Universal Robots PolyScope program: Bridge_triangle_roof.urp

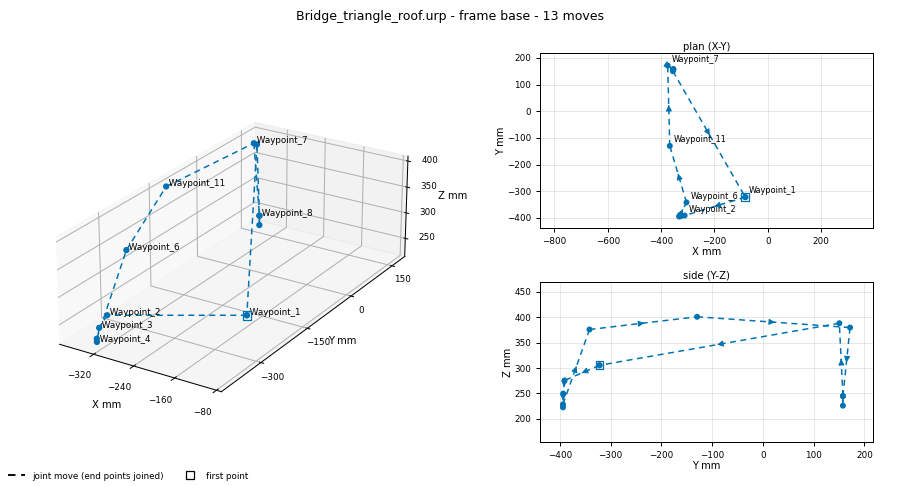
[picture p0: tool path of Bridge_triangle_roof.urp in frame base, 13 of 13 moves have a stored position in this frame; points joined in program order, loops and branches not executed]
Program Bridge_triangle_roof (installation=default directory=/programs/usbdisk/Zahra createdIn=5.11.11.1010533 lastSavedIn=5.11.11.1010533 robotSerialNumber=20205300864)
Calibrated DH parameters: a=[-0.000166, -0.243494, -0.153108, 0.000057, -0.000123, 0]; d=[0.151897, -1.34267, 53.988124, -52.514559, 0.085283, 0.092193]; alpha=[1.572472, -0.003756, 0.002824, 1.570807, -1.572621, 0]; deltaTheta=[0, 0.020704, 7.033215, -0.770746, 0.000004, 0]
Robot Program (runOnlyOnce=true)
  MoveJ speed 60 deg/s, acceleration 80 deg/s^2 (useActiveTCP=true) feature=Base
    Waypoint Waypoint_1: TCP in base x=-84.299 y=-321.875 z=305.481 mm, rx=-2.0809 ry=-2.2572 rz=0.0984 rad; joints [-79.978, -91.201, -87.971, -91.7, 84.671, 815.506] deg
    Waypoint Waypoint_2: TCP in base x=-311.801 y=-390.806 z=275.565 mm, rx=-2.2649 ry=-2.1055 rz=0.1333 rad; joints [-112.548, -138.493, -28.193, -99.813, 85.37, 791.491] deg
    Waypoint Waypoint_3: TCP in base x=-326.771 y=-393.435 z=249.787 mm, rx=2.215 ry=2.2214 rz=-0.0644 rad; joints [-114.765, -143.708, -24.768, -99.132, 89.224, 785.045] deg
    Waypoint Waypoint_4: TCP in base x=-331.937 y=-393.874 z=222.59 mm, rx=2.1803 ry=2.2287 rz=-0.0042 rad; joints [-115.635, -145.452, -28.079, -95.78, 91.072, 783.114] deg
    URCap Gripper (Robotiq_Grippers, Robotiq Inc.) dataModel(position=59.2156862745098, force=94.0, speed=40.0, positionInDouble=59.2156862745098, forceInDouble=94.0, speedInDouble=40.0, slaveIds=[9], blocking=true, robotCompliant=false)
    Waypoint Waypoint_5: TCP in base x=-331.939 y=-393.873 z=228.535 mm, rx=2.1803 ry=2.2287 rz=-0.0043 rad; joints [-115.63, -145.851, -25.689, -97.768, 91.067, 783.115] deg
    Waypoint Waypoint_6: TCP in base x=-304.837 y=-341.621 z=375.948 mm, rx=2.1229 ry=2.1896 rz=-0.3358 rad; joints [-115.077, -126.752, -25.522, -104.372, 89.719, 783.12] deg
    Waypoint Waypoint_11: TCP in base x=-367.481 y=-129.683 z=400.982 mm, rx=-2.0842 ry=-2.3405 rz=-0.0182 rad; joints [-140.769, -116.62, -27.668, -126.196, 89.307, 752.639] deg
    Waypoint Waypoint_7: TCP in base x=-375.414 y=171.565 z=379.774 mm, rx=-2.1093 ry=-2.3182 rz=0.0687 rad; joints [-186.479, -119.065, -31.593, -117.454, 91.662, 708.179] deg
    Waypoint Waypoint_8: TCP in base x=-354.29 y=157.579 z=244.826 mm, rx=-2.2211 ry=-2.2068 rz=0.0358 rad; joints [-184.497, -106.857, -86.723, -75.009, 90.588, 716.008] deg
    Waypoint Waypoint_9: TCP in base x=-354.309 y=157.557 z=225.911 mm, rx=-2.2211 ry=-2.2068 rz=0.0359 rad; joints [-184.501, -108.084, -90.347, -70.153, 90.592, 716.013] deg
    URCap Gripper (Robotiq_Grippers, Robotiq Inc.) dataModel(position=33.72549019607843, force=94.0, speed=40.0, positionInDouble=33.72549019607843, forceInDouble=94.0, speedInDouble=40.0, slaveIds=[9], blocking=true, robotCompliant=false)
    Waypoint Waypoint_8: TCP in base x=-354.29 y=157.579 z=244.826 mm, rx=-2.2211 ry=-2.2068 rz=0.0358 rad; joints [-184.497, -106.857, -86.723, -75.009, 90.588, 716.008] deg
    Waypoint Waypoint_10: TCP in base x=-355.906 y=150.496 z=388.296 mm, rx=-2.1322 ry=-2.1758 rz=0.1564 rad; joints [-183.387, -106.861, -50.233, -105.001, 90.897, 715.571] deg
    Waypoint Waypoint_1: TCP in base x=-84.299 y=-321.875 z=305.481 mm, rx=-2.0809 ry=-2.2572 rz=0.0984 rad; joints [-79.978, -91.201, -87.971, -91.7, 84.671, 815.506] deg
